FUNCTION_BLOCK InductiveSensor IMPLEMENTS ITF_BinarySensor
VAR_INPUT
END_VAR
VAR_OUTPUT
END_VAR
VAR
	//Hardware
	DI_WPMetallic AT %I* : BOOL;
END_VAR

PROPERTY Value : BOOL
GET
Value := DI_WPMetallic;
END_GET
END_PROPERTY

END_FUNCTION_BLOCK

(* stored: Version 1.1.0.1
   POU InductiveSensor: Id {4736a843-aa8d-4180-a544-b4f7627b75c7}, SpecialFunc None
   Property Value: Id {e845cd24-491d-4a7b-a604-a16b20849302}
   Get Get: Id {58c9b07c-205a-494d-b0a6-609f4e2d84e3} *)
